# EPICS substitutions: evrMrmApp/Db/PSI/evr-pmc-230.substitutions
# Record set for a PMC-EVR-230
#
# Macros:
#  EVR = Card name (same as mrmEvrSetupPCI())
#  SYS = System name (ie SR-TM)
#
# Record names have the general forms:
#  $(SYS)-$(EVR):Signal-SD

file "evrBase.db"
{pattern
{P, OBJ, EVNT1HZ}
{"$(SYS)-$(EVR):", $(EVR), 125}
}

file "sfp.db"
{
{P="$(SYS)-$(EVR):SFP-", OBJ="$(EVR):SFP"}
}

file "evrScale.db"
{pattern
{IDX, P, SN, OBJ, MAX}
{0, "$(SYS)-$(EVR):", "$(SYS)-$(EVR):PS-$(IDX)-", "$(EVR):PS$(IDX)", "0xffff"}
{1, "$(SYS)-$(EVR):", "$(SYS)-$(EVR):PS-$(IDX)-", "$(EVR):PS$(IDX)", "0xffff"}
{2, "$(SYS)-$(EVR):", "$(SYS)-$(EVR):PS-$(IDX)-", "$(EVR):PS$(IDX)", "0xffff"}
}

# Pulse generators w/o a prescaler set NOPS=1
file "evrPulser.db"
{pattern
{PID, P, PN, OBJ, DMAX, WMAX, PMAX, NOPS}
{0, "$(SYS)-$(EVR):", "$(SYS)-$(EVR):DlyGen-$(PID)-", "$(EVR):Pul$(PID)", "0xffffff", "0xffff", "0xff", 0}
{1, "$(SYS)-$(EVR):", "$(SYS)-$(EVR):DlyGen-$(PID)-", "$(EVR):Pul$(PID)", "0xffffff", "0xffff", "0xff", 0}
{2, "$(SYS)-$(EVR):", "$(SYS)-$(EVR):DlyGen-$(PID)-", "$(EVR):Pul$(PID)", "0xffffff", "0xffff", "0xff", 0}
{3, "$(SYS)-$(EVR):", "$(SYS)-$(EVR):DlyGen-$(PID)-", "$(EVR):Pul$(PID)", "0xffffff", "0xffff", "0xff", 0}
{4, "$(SYS)-$(EVR):", "$(SYS)-$(EVR):DlyGen-$(PID)-", "$(EVR):Pul$(PID)", "0xffffff", "0xffff", "1", 1}
{5, "$(SYS)-$(EVR):", "$(SYS)-$(EVR):DlyGen-$(PID)-", "$(EVR):Pul$(PID)", "0xffffff", "0xffff", "1", 1}
{6, "$(SYS)-$(EVR):", "$(SYS)-$(EVR):DlyGen-$(PID)-", "$(EVR):Pul$(PID)", "0xffffff", "0xffff", "1", 1}
{7, "$(SYS)-$(EVR):", "$(SYS)-$(EVR):DlyGen-$(PID)-", "$(EVR):Pul$(PID)", "0xffffff", "0xffff", "1", 1}
{8, "$(SYS)-$(EVR):", "$(SYS)-$(EVR):DlyGen-$(PID)-", "$(EVR):Pul$(PID)", "0xffffff", "0xffff", "1", 1}
{9, "$(SYS)-$(EVR):", "$(SYS)-$(EVR):DlyGen-$(PID)-", "$(EVR):Pul$(PID)", "0xffffff", "0xffff", "1", 1}
}

# Default to 3 possible trigger mappings per pulser
file "evrPulsermap.db"
{pattern
{PID, NAME, OBJ, F, EVT}
{0, "$(SYS)-$(EVR):DlyGen-$(PID)-Evt-Trig0-SP", "$(EVR):Pul$(PID)", Trig, 0}
{0, "$(SYS)-$(EVR):DlyGen-$(PID)-Evt-Trig1-SP", "$(EVR):Pul$(PID)", Trig, 0}
{0, "$(SYS)-$(EVR):DlyGen-$(PID)-Evt-Trig2-SP", "$(EVR):Pul$(PID)", Trig, 0}
{1, "$(SYS)-$(EVR):DlyGen-$(PID)-Evt-Trig0-SP", "$(EVR):Pul$(PID)", Trig, 0}
{1, "$(SYS)-$(EVR):DlyGen-$(PID)-Evt-Trig1-SP", "$(EVR):Pul$(PID)", Trig, 0}
{1, "$(SYS)-$(EVR):DlyGen-$(PID)-Evt-Trig2-SP", "$(EVR):Pul$(PID)", Trig, 0}
{2, "$(SYS)-$(EVR):DlyGen-$(PID)-Evt-Trig0-SP", "$(EVR):Pul$(PID)", Trig, 0}
{2, "$(SYS)-$(EVR):DlyGen-$(PID)-Evt-Trig1-SP", "$(EVR):Pul$(PID)", Trig, 0}
{2, "$(SYS)-$(EVR):DlyGen-$(PID)-Evt-Trig2-SP", "$(EVR):Pul$(PID)", Trig, 0}
{3, "$(SYS)-$(EVR):DlyGen-$(PID)-Evt-Trig0-SP", "$(EVR):Pul$(PID)", Trig, 0}
{3, "$(SYS)-$(EVR):DlyGen-$(PID)-Evt-Trig1-SP", "$(EVR):Pul$(PID)", Trig, 0}
{3, "$(SYS)-$(EVR):DlyGen-$(PID)-Evt-Trig2-SP", "$(EVR):Pul$(PID)", Trig, 0}
{4, "$(SYS)-$(EVR):DlyGen-$(PID)-Evt-Trig0-SP", "$(EVR):Pul$(PID)", Trig, 0}
{4, "$(SYS)-$(EVR):DlyGen-$(PID)-Evt-Trig1-SP", "$(EVR):Pul$(PID)", Trig, 0}
{4, "$(SYS)-$(EVR):DlyGen-$(PID)-Evt-Trig2-SP", "$(EVR):Pul$(PID)", Trig, 0}
{5, "$(SYS)-$(EVR):DlyGen-$(PID)-Evt-Trig0-SP", "$(EVR):Pul$(PID)", Trig, 0}
{5, "$(SYS)-$(EVR):DlyGen-$(PID)-Evt-Trig1-SP", "$(EVR):Pul$(PID)", Trig, 0}
{5, "$(SYS)-$(EVR):DlyGen-$(PID)-Evt-Trig2-SP", "$(EVR):Pul$(PID)", Trig, 0}
{6, "$(SYS)-$(EVR):DlyGen-$(PID)-Evt-Trig0-SP", "$(EVR):Pul$(PID)", Trig, 0}
{6, "$(SYS)-$(EVR):DlyGen-$(PID)-Evt-Trig1-SP", "$(EVR):Pul$(PID)", Trig, 0}
{6, "$(SYS)-$(EVR):DlyGen-$(PID)-Evt-Trig2-SP", "$(EVR):Pul$(PID)", Trig, 0}
{7, "$(SYS)-$(EVR):DlyGen-$(PID)-Evt-Trig0-SP", "$(EVR):Pul$(PID)", Trig, 0}
{7, "$(SYS)-$(EVR):DlyGen-$(PID)-Evt-Trig1-SP", "$(EVR):Pul$(PID)", Trig, 0}
{7, "$(SYS)-$(EVR):DlyGen-$(PID)-Evt-Trig2-SP", "$(EVR):Pul$(PID)", Trig, 0}
{8, "$(SYS)-$(EVR):DlyGen-$(PID)-Evt-Trig0-SP", "$(EVR):Pul$(PID)", Trig, 0}
{8, "$(SYS)-$(EVR):DlyGen-$(PID)-Evt-Trig1-SP", "$(EVR):Pul$(PID)", Trig, 0}
{8, "$(SYS)-$(EVR):DlyGen-$(PID)-Evt-Trig2-SP", "$(EVR):Pul$(PID)", Trig, 0}
{9, "$(SYS)-$(EVR):DlyGen-$(PID)-Evt-Trig0-SP", "$(EVR):Pul$(PID)", Trig, 0}
{9, "$(SYS)-$(EVR):DlyGen-$(PID)-Evt-Trig1-SP", "$(EVR):Pul$(PID)", Trig, 0}
{9, "$(SYS)-$(EVR):DlyGen-$(PID)-Evt-Trig2-SP", "$(EVR):Pul$(PID)", Trig, 0}
}

file "evrIn.db"
{pattern
{IN, OBJ, DESC}
{"$(SYS)-$(EVR):In-0-", "$(EVR):FPIn0", "EXT IN (TTL)"}
}

file "evrOut.db"
{pattern
{ON, OBJ, DESC}
{"$(SYS)-$(EVR):Out-FP0-", "$(EVR):FrontOut0", "OUT0 (TTL)"}
{"$(SYS)-$(EVR):Out-FP1-", "$(EVR):FrontOut1", "OUT1 (TTL)"}
{"$(SYS)-$(EVR):Out-FP2-", "$(EVR):FrontOut2", "OUT2 (TTL)"}
}
